# EPICS StreamDevice protocol: aeroflexSup/aeroflex_2023A.proto
InTerminator = '\n';
OutTerminator = '\n';

getCarrierFrequency {
	out "CFRQ?";
	in ":CFRQ:VALUE %f;INC %*f;MODE %*s";
}

setModulation {
	out "MODE %{FM,AM,PULSE|FM,AM|PM,AM,PULSE|PM,AM|AM,PULSE|AM|FM,PULSE|FM|PM,PULSE|PM|FSK2L,PULSE|FSK2L|FSK4L}";
}
